FUNCTION_BLOCK FB_Moteur
VAR_INPUT
	fbPower: MC_power;
	fbMoveAbsolute: MC_MoveAbsolute;
	fbHome: MC_Home;
	fbReset: MC_Reset;
END_VAR
VAR_OUTPUT
END_VAR
VAR
	
END_VAR
VAR_IN_OUT
	fbAxe: AXIS_REF;
END_VAR

fbPower(Axis:=fbAxe);
fbMoveAbsolute(Axis:=fbAxe);
fbHome(Axis:=fbAxe);
fbReset(Axis:=fbAxe);

END_FUNCTION_BLOCK

(* stored: Version 1.1.0.1, ProductVersion 3.1.4020.12
   POU FB_Moteur: Id {c2c97c00-92e1-48e6-ab83-9956cf4b0348}, SpecialFunc None *)
